// TIA Portal project "Trabajo_Automatización" (V18)

(* hardware
DEVICE "S7-1500/ET200MP station_1"  S7-1500 station
   slot 0: "Rail_0"  Rack  6ES7 590-1***0-0AA0
   slot 1: "PLC_1"  Unspecific CPU 1500  6ES7 5XX-XXXXX-XXXX  V3.0
*)

// ===== PLC "PLC_1"  Unspecific CPU 1500 =====

FUNCTION_BLOCK "ciclo"   // FB1, STL
TITLE = Gestiona una maniobra de la pick and place (carga o descarga)
{ S7_Optimized_Access := 'TRUE' }
VERSION : 0.1
// el control emplea dos instancias
// Maniobra compuesta por una secuencia de 3 acciones de control
// No tiene gestion de errores
// Se emplea plantilla de macroetapa para la implementacion
   VAR_INPUT
      lectura_correcta : Bool;   // finalización de la identificación
      escritura_correcta : Bool;   // finalización de la actualización del estado del producto
      fin_maniobra : Bool;   // finalización de la maniobra de la Pick&Place
      OK_reposo : Bool;   // confirmación del reposo
   END_VAR
   VAR_OUTPUT
      Bit_finalización : Bool;   // informa de finalizacion correcta (XSALIDA:=TRUE)
   END_VAR
   VAR_IN_OUT
      lectura : Bool;   // identificación del producto y su estado
      escritura : Bool;   // escritura del estado del producto agarrado
      maniobra : Bool;   // acción que debe ejecutar la Pick&Place
      reposo : Bool;   // vuelta al reposo de la Pick&Place
   END_VAR
   VAR
      Bit_trabajo : Bool;   // Static para no perder la memoria entre estados
      X1 : Bool;   // lectura en ejecución
      X2 : Bool;   // escritura en ejecución
      X3 : Bool;   // acción en ejecución
      X4 : Bool;   // señal de reposo
      XSALIDA : Bool;   // etapa de salida finalizacion correcta de la macro
   END_VAR
BEGIN

REGION Network 1: desconexion del grafcet GE encapsulado por M<#id>
         A     #XSALIDA;  //estado de salida

         R     #XSALIDA;  //necesario anularlo. si se llama en el futuro debe estar desconectado;
   //    no se puede modificar desde fuera

         R     #Bit_trabajo;  //para poder arrancar en el futuro
         S     #Bit_finalización;  //aviso hacia el exterior del final de la macro

         R     #lectura;
         R     #escritura;
         R     #maniobra;
         R     #reposo;

         BEC;  //fin de bloque condicionado a XSALIDA
   //    el usuario no debe llamar al bloque en el mismo ciclo en el que el bloque finaliza.
END_REGION

REGION Network 2: arranque del grafcet encapsulado en M<#id>
         SET;  //RLO:=TRUE - tautologia. Independencia de eventos de fuera
         FP    #Bit_trabajo;  // evento de arranque. En cuanto se llama al bloque, arranca el ciclo.
   //Pasa de 0 a 1 y se queda en 1 mientras el bloque está operativo.

         R     #Bit_finalización;  //OBLIGATORIO

   //activacion estado inicial de GE. No sería necesario limpiar los estados al finalizar (redundancia)
         S     #X1;
         R     #X2;
         R     #X3;
         R     #X4;
         R     #XSALIDA;
END_REGION

REGION Network 3: lectura en ejecución
         A     #X1;
         A     #lectura_correcta;
         S     #X2;
         R     #X1;
END_REGION

REGION Network 4: escritura en ejecucion
         A     #X2;
         A     #escritura_correcta;
         S     #X3;
         R     #X2;
END_REGION

REGION Network 5: acción en ejecución
         A     #X3;
         A     #fin_maniobra;
         S     #X4;
         R     #X3;
END_REGION

REGION Network 6: señal de reposo
         A     #X4;
         A     #OK_reposo;
         S     #XSALIDA;
         R     #X4;
END_REGION

REGION Network 7: tratamiento maniobra primera
         A     #X1;
         =     #lectura;
END_REGION

REGION Network 8: tratamiento maniobra segunda
         A     #X2;
         =     #escritura;
END_REGION

REGION Network 9: tratamiento maniobra tercera
         A     #X3;
         =     #maniobra;
END_REGION

REGION Network 10: tratamiento maniobra cuarta
         A     #X4;
         =     #reposo;
END_REGION
END_FUNCTION_BLOCK

FUNCTION_BLOCK "proceso"   // FB2, STL
TITLE = Gestiona una maniobra de la pick and place (carga o descarga)
{ S7_Optimized_Access := 'TRUE' }
VERSION : 0.1
// el control emplea dos instancias
// Maniobra compuesta por una secuencia de 3 acciones de control
// No tiene gestion de errores
// Se emplea plantilla de macroetapa para la implementacion
   VAR_INPUT
      A_disponible : Bool;   // espacio disponible en el lado A
      B_disponible : Bool;   // espacio disponible en el lado B
      lectura_correcta : Bool;
      escritura_correcta : Bool;
      fin_maniobra : Bool;
      OK_reposo : Bool;   // confirmación del reposo
   END_VAR
   VAR_OUTPUT
      Bit_finalización : Bool;   // informa de finalizacion correcta (XSALIDA:=TRUE)
   END_VAR
   VAR_IN_OUT
      RFID_Estacion_A : Bool;
      Interaccion_Cinta_Estacion_A : Bool;
      RFID_Estacion_B : Bool;
      Interaccion_Cinta_Estacion_B : Bool;
      RFID_Post : Bool;
      reposo : Bool;   // vuelta al reposo de la Pick&Place
   END_VAR
   VAR
      Bit_trabajo : Bool;   // Static para no perder la memoria entre estados
      IN : Bool;   // estado de espera
      XA : Bool;   // ciclo por lado A
      XB : Bool;   // ciclo por lado B
      ciclo_Estación_A : "ciclo";
      ciclo_Estación_B : "ciclo";
      defecto : Bool;   // sin disponibilidad. no ejecutar maniobra
      XSALIDA : Bool;   // etapa de salida finalizacion correcta de la macro
   END_VAR
BEGIN

REGION Network 1: desconexion del grafcet GE encapsulado por M<#id>
         A     #XSALIDA;  //estado de salida

         R     #XSALIDA;  //necesario anularlo. si se llama en el futuro debe estar desconectado;
   //    no se puede modificar desde fuera

         R     #Bit_trabajo;  //para poder arrancar en el futuro
         S     #Bit_finalización;  //aviso hacia el exterior del final de la macro

         R     #reposo;

         BEC;  //fin de bloque condicionado a XSALIDA
   //    el usuario no debe llamar al bloque en el mismo ciclo en el que el bloque finaliza.
END_REGION

REGION Network 2: arranque del grafcet encapsulado en M<#id>
         SET;  //RLO:=TRUE - tautologia. Independencia de eventos de fuera
         FP    #Bit_trabajo;  // evento de arranque. En cuanto se llama al bloque, arranca el ciclo.
   //Pasa de 0 a 1 y se queda en 1 mientras el bloque está operativo.

         R     #Bit_finalización;  //OBLIGATORIO

   //activacion estado inicial de GE. No sería necesario limpiar los estados al finalizar (redundancia)
         S     #XA;
         R     #XB;
         R     #defecto;
         R     #XSALIDA;
END_REGION

REGION Network 3: evaluación disponibilidad del lado A
         A     #IN;
         A     #A_disponible;
         S     #XA;
         R     #IN;
END_REGION

REGION Network 4: evaluación disponibilidad del lado B
         A     #IN;
         A     #B_disponible;
         S     #XB;
         R     #IN;
END_REGION

REGION Network 5: evaluación del defecto
         A     #IN;
         AN    #A_disponible;
         AN    #B_disponible;
         S     #defecto;
         R     #IN;
END_REGION

REGION Network 6: tratamiento interacción estación A y cinta
         A     #XA;
         JCN   _000;
         CALL  #ciclo_Estación_A
         ( lectura_correcta   := #lectura_correcta,
           escritura_correcta := #escritura_correcta,
           fin_maniobra       := #fin_maniobra,
           OK_reposo          := #OK_reposo,
           Bit_finalización   := #Bit_finalización,
           lectura            := #RFID_Estacion_A,
           escritura          := #RFID_Post_Estacion_A,
           maniobra           := #Interaccion_Cinta_Estacion_A,
           reposo             := #reposo
         );

   //TODO@EMER y rearme
   //TODO@gestión de errores
         A     #ciclo_Estación_A.Bit_finalización;
         S     #XSALIDA;
         R     #XA;
   _000: NOP   0;
END_REGION

REGION Network 7: tratamiento interaccion estación B y cinta
         A     #XB;
         JCN   _001;
         CALL  #ciclo_Estación_B
         ( lectura_correcta   := #lectura_correcta,
           escritura_correcta := #escritura_correcta,
           fin_maniobra       := #fin_maniobra,
           OK_reposo          := #OK_reposo,
           Bit_finalización   := #Bit_finalización,
           lectura            := #RFID_Estacion_B,
           escritura          := #RFID_Post,
           maniobra           := #Interaccion_Cinta_Estacion_B,
           reposo             := #reposo
         );

   //TODO@EMER y rearme
   //TODO@gestión de errores
         A     #ciclo_Estación_B.Bit_finalización;
         S     #XSALIDA;
         R     #XB;
   _001: NOP   0;
END_REGION

REGION Network 8: tratamiento defecto
         A     #defecto;
         =     #reposo;
END_REGION

REGION Network 9: fin defecto
         A     #OK_reposo;
         R     #defecto;
         S     #XSALIDA;
END_REGION
END_FUNCTION_BLOCK

FUNCTION_BLOCK "Pick&Place"   // FB3, STL
{ S7_Optimized_Access := 'TRUE' }
VERSION : 0.1
   VAR_INPUT
      OK_AUTO : Bool;
      OK_HOME : Bool;
      S_Caja_Vacia_C1 : Bool;
      S_Caja_Vacia_C2 : Bool;
      S_Caja_C1 : Bool;
      S_Caja_C2 : Bool;
   END_VAR
   VAR_OUTPUT
      bit_fin : Bool;
   END_VAR
   VAR_IN_OUT
      AUTODIAG : Bool;
      HOME : Bool;
   END_VAR
   VAR
      X0 : Bool;   // autodiagnóstico de encendido
      X1 : Bool;   // señal de reposo
      X2 : Bool;   // standby
      defecto : Bool;
      proceso_Descarga_C1 : "proceso";
   END_VAR
BEGIN

REGION Network 1: standby
         A     #X2;
         A     #S_Caja_Vacia_C1;
         JCN   _000;
         CALL  #proceso_Descarga_C1
         ( A_disponible                 := A_disponible,
           B_disponible                 := B_disponible,
           lectura_correcta             := OK_READ,
           escritura_correcta           := OK_WRITE,
           fin_maniobra                 := fin_maniobra,
           OK_reposo                    := #OK_HOME,
           Bit_finalización             := #bit_fin,
           RFID_Estacion_A              := RFID_FROM_SA,
           Interaccion_Cinta_Estacion_A := FROM_C1_TO_SA,
           RFID_Estacion_B              := RFID_FROM_SB,
           Interaccion_Cinta_Estacion_B := FROM_C1_TO_SB,
           RFID_Post                    := RFID_SET,
           reposo                       := #HOME
         );

   //TODO@EMER y rearme
   //TODO@gestión de errores
         A     #proceso_Descarga_C1.Bit_finalización;
         S     #X2;
         R     #XEspera;
   _000: NOP   0;
END_REGION

REGION Network 2
         A     #X2;
         A     #S_Caja_Vacia_C2;
END_REGION
END_FUNCTION_BLOCK

ORGANIZATION_BLOCK "Main"   // OB1, STL, ProgramCycle
TITLE = "Main Program Sweep (Cycle)"
{ S7_Optimized_Access := 'TRUE' }
VERSION : 0.1
   VAR_INPUT
      Initial_Call : Bool;   // Initial call of this OB
      Remanence : Bool;   // =True, if remanent data are available
   END_VAR
BEGIN
END_ORGANIZATION_BLOCK